(* IEC 61131-3 sources: AXOpen/src/components.dukane.welders/ctrl/src/Axo_IQ_SeriesWelder (part 6) *)

                    IF TRUE THEN
                        THIS.CallTimers(FALSE);
                        _progress := 474;
                    END_IF;
                END_IF;

                IF _progress = 474 THEN                                                                                     // TemplateTask_20steps_6 running: , <add the detailed description of the current action 15>
                    IF _infoTimer.output THEN
                        TaskMessenger.Activate( UINT#674, eAxoMessageCategory#Warning);
                        Status.Error.Id :=      UINT#674;
                    END_IF;

                    IF TRUE THEN
                        THIS.CallTimers(FALSE);
                        _progress := 475;
                    END_IF;
                END_IF;

                IF _progress = 475 THEN                                                                                     // TemplateTask_20steps_6 running: , <add the detailed description of the current action 16>
                    IF _infoTimer.output THEN
                        TaskMessenger.Activate( UINT#675, eAxoMessageCategory#Warning);
                        Status.Error.Id :=      UINT#675;
                    END_IF;

                    IF TRUE THEN
                        THIS.CallTimers(FALSE);
                        _progress := 476;
                    END_IF;
                END_IF;

                IF _progress = 476 THEN                                                                                     // TemplateTask_20steps_6 running: , <add the detailed description of the current action 17>
                    IF _infoTimer.output THEN
                        TaskMessenger.Activate( UINT#676, eAxoMessageCategory#Warning);
                        Status.Error.Id :=      UINT#676;
                    END_IF;

                    IF TRUE THEN
                        THIS.CallTimers(FALSE);
                        _progress := 477;
                    END_IF;
                END_IF;

                IF _progress = 477 THEN                                                                                     // TemplateTask_20steps_6 running: , <add the detailed description of the current action 18>
                    IF _infoTimer.output THEN
                        TaskMessenger.Activate( UINT#677, eAxoMessageCategory#Warning);
                        Status.Error.Id :=      UINT#677;
                    END_IF;

                    IF TRUE THEN
                        THIS.CallTimers(FALSE);
                        _progress := 478;
                    END_IF;
                END_IF;

                IF _progress = 478 THEN                                                                                     // TemplateTask_20steps_6 running: , <add the detailed description of the current action 19>
                    IF _infoTimer.output THEN
                        TaskMessenger.Activate( UINT#678, eAxoMessageCategory#Warning);
                        Status.Error.Id :=      UINT#678;
                    END_IF;

                    IF TRUE THEN
                        THIS.CallTimers(FALSE);
                        _progress := 479;
                    END_IF;
                END_IF;

                IF _progress = 479 THEN                                                                                     // TemplateTask_20steps_6 running: , <add the detailed description of the current action 20>
                    TemplateTask_20steps_6.DoneWhen(TRUE);
                    _progress := 0;
                END_IF;

                THIS.CallTimers(TRUE);

                TemplateTask_20steps_6.ThrowWhen(_errorTimer.output);
                Status.Action.Id := TO_UINT(_progress);
                TemplateTask_20steps_6.ThrowWhen(TemplateTask_20steps_6.Duration >= Config.TaskTimeout AND Config.TaskTimeout > T#0s ,'TemplateTask_20steps_6 timeout.');
            END_IF;
            IF TemplateTask_20steps_6.DoneReached() THEN
                Status.Action.Id :=  UINT#261;
                Status.Error.Id :=  UINT#0;
            ELSIF TemplateTask_20steps_6.ErrorOccured() THEN
                Status.Action.Id :=  UINT#10160;
                Status.Error.Id  :=  UINT#10160;
            ELSIF TemplateTask_20steps_6.AbortTriggered()THEN
                Status.Action.Id :=  UINT#10161;
                Status.Error.Id  :=  UINT#10161;
            END_IF;
            Messenger.ActivateOnCondition(ULINT#10160,TemplateTask_20steps_6.HasError(), eAxoMessageCategory#Error);
            Messenger.ActivateOnCondition(ULINT#10161,TemplateTask_20steps_6.IsAborted(), eAxoMessageCategory#Error);
            Messenger.ActivateOnCondition(ULINT#262,TemplateTask_20steps_6.RestoreTriggered() , eAxoMessageCategory#Error);
            IF TemplateTask_20steps_6.RestoreTriggered() AND _progress >= 460 AND _progress <= 479  THEN
                Status.Action.Id :=  UINT#262;
                _progress := 0;
            END_IF;
            //******************************************

            //***********Update outputs ****************
            // ============================================================================
            // Network 14: Write synchronous data to the module (outputs)
            // ============================================================================
            // This was original outputs writing =>
            // synchronous_write_retval := DPWR_DAT(LADDR := outputs_hw_id,RECORD := iq_if._out);
            // <= This was original outputs writing

            // This is new outputs writing =>
            _data_out[0].%X0    :=  Outputs.N0;
            _data_out[0].%X1    :=  Outputs.N01;
            _data_out[0].%X2    :=  Outputs.N02;
            _data_out[0].%X3    :=  Outputs.N03;
            _data_out[0].%X4    :=  Outputs.N04;
            _data_out[0].%X5    :=  Outputs.N05;
            _data_out[0].%X6    :=  Outputs.N06;
            _data_out[0].%X7    :=  Outputs.ClearSetup;
            _data_out[1].%X0    :=  Outputs.N2;
            _data_out[1].%X1    :=  Outputs.N3;
            _data_out[1].%X2    :=  Outputs.N4;
            _data_out[1].%X3    :=  Outputs.N5;
            _data_out[1].%X4    :=  Outputs.N6;
            _data_out[1].%X5    :=  Outputs.N7;
            _data_out[1].%X6    :=  Outputs.N8;
            _data_out[1].%X7    :=  Outputs.N9;
            _data_out[2].%X0    :=  Outputs.RunScan;
            _data_out[2].%X1    :=  Outputs.N11;
            _data_out[2].%X2    :=  Outputs.N12;
            _data_out[2].%X3    :=  Outputs.N13;
            _data_out[2].%X4    :=  Outputs.N14;
            _data_out[2].%X5    :=  Outputs.N15;
            _data_out[2].%X6    :=  Outputs.N16;
            _data_out[2].%X7    :=  Outputs.N17;
            _data_out[3].%X0    :=  Outputs.RunContinuously;
            _data_out[3].%X1    :=  Outputs.RunWeld;
            _data_out[3].%X2    :=  Outputs.RunTest;
            _data_out[3].%X3    :=  Outputs.ClearError;
            _data_out[3].%X4    :=  Outputs.OTF_AmplitudeEnable;
            _data_out[3].%X5    :=  Outputs.CycleStop;
            _data_out[3].%X6    :=  Outputs.FrontPanelLockout_0;
            _data_out[3].%X7    :=  Outputs.FrontPanelLockout_1;

            tmp_DW              :=  TO_DWORD(Outputs.OTF_Amp_Setpoint);
            _data_out[4]        :=  tmp_DW.%B3;
            _data_out[5]        :=  tmp_DW.%B2;
            _data_out[6]        :=  tmp_DW.%B1;
            _data_out[7]        :=  tmp_DW.%B0;

            tmp_DW              :=  TO_DWORD(Outputs.ActiveSetupSelection);
            _data_out[8]        :=  tmp_DW.%B3;
            _data_out[9]        :=  tmp_DW.%B2;
            _data_out[10]       :=  tmp_DW.%B1;
            _data_out[11]       :=  tmp_DW.%B0;

            tmp_DW              :=  TO_DWORD(Outputs.RunningSetupSelection);
            _data_out[12]       :=  tmp_DW.%B3;
            _data_out[13]       :=  tmp_DW.%B2;
            _data_out[14]       :=  tmp_DW.%B1;
            _data_out[15]       :=  tmp_DW.%B0;

            tmp_DW              :=  TO_DWORD(Outputs.RunningMPCProbeSelection);
            _data_out[16]       :=  tmp_DW.%B3;
            _data_out[17]       :=  tmp_DW.%B2;
            _data_out[18]       :=  tmp_DW.%B1;
            _data_out[19]       :=  tmp_DW.%B0;

            synchronous_write_retval := TO_INT(WriteData(LADDR := TO_WORD(Config.HWIDs.HwID_PLC_to_iQ_Outputs),RECORD := _data_out));
            IF synchronous_write_retval > INT#0 THEN
                Messenger.Activate(UINT#1231, eAxoMessageCategory#ProgrammingError);
                Status.Error.Id := UINT#1231;
                RETURN;
            END_IF;
            // <= This is new outputs writing

            // ============================================================================
            // Network 15: Read req - HMI export (indicators)
            // ============================================================================
            // tof_async_read_ind(IN := (par_read_map <> 0) OR (on_demand_read_map <> 0) OR (model_read_map <> 0),PT := T#500ms);
            // Hmi.s.AsyncReadIndicator := tof_async_read_ind.Q;
            tof_async_read_ind(signal := (par_read_map <> WORD#0) OR (on_demand_read_map <> WORD#0) OR (model_read_map <> WORD#0) , duration := T#500ms);
            Hmi.s.AsyncReadIndicator := tof_async_read_ind.output;

            // ============================================================================
            // Network 16: Read acyclic data
            // ============================================================================
            //Try asynchronous comunication only when synchronous comunication is stable (no errors for 1s)
            // IF (coms_stable) THEN

            //     //Save rd_req value from previous iteation
            //     prev_rd_req := ReadRecord.request;

            //     // Proces valid data if needed
            //     IF ReadRecord.VALID THEN
            //         Hmi.read_status[async_read_no] := ReadRecord.STATUS;
            //         CASE async_read_no OF
            //             -16: // Model no decode to string
            //                 // Chars_TO_Strg(Chars := str_read_buffer,
            //                 //               pChars := 0,
            //                 //               Cnt := RD_REC.length,
            //                 //               Strg => ModelInfo.ModelNumber);
            //                 _data_255[0]:= TO_BYTE(ReadRecord.length);
            //                 FOR index := UINT#0 TO ReadRecord.length DO
            //                     _data_255[index + UINT#1] := str_read_buffer_254[index];
            //                 END_FOR;
            //                 Deserialize(UDINT#0, str_read_buffer_254, ModelInfo.ModelNumber);

            //             -15:
            //                 Deserialize(UDINT#0, str_read_buffer_254, ModelInfo.SerialNumber);

            //             -14: // MB firmware version decode to string
            //                 // Chars_TO_Strg(Chars := str_read_buffer_254,
            //                 //               pChars := 0,
            //                 //               Cnt := RD_REC.length,
            //                 //               Strg => ModelInfo.MB_FirmwareVersion);
            //                 _data_255[0]:= TO_BYTE(ReadRecord.length);
            //                 FOR index := UINT#0 TO ReadRecord.length DO
            //                     _data_255[index + UINT#1] := str_read_buffer_254[index];
            //                 END_FOR;
            //                 Deserialize(UDINT#0, str_read_buffer_254, ModelInfo.MB_FirmwareVersion);

            //             -13: // FP firmware version decode to string
            //                 // Chars_TO_Strg(Chars := str_read_buffer_254,
            //                 //               pChars := 0,
            //                 //               Cnt := RD_REC.length,
            //                 //               Strg => ModelInfo.FP_FirmwareVersion);
            //                 _data_255[0]:= TO_BYTE(ReadRecord.length);
            //                 FOR index := UINT#0 TO ReadRecord.length DO
            //                     _data_255[index + UINT#1] := str_read_buffer_254[index];
            //                 END_FOR;
            //                 Deserialize(UDINT#0, str_read_buffer_254, ModelInfo.FP_FirmwareVersion);

            //             -12: // MB bootloader version decode to string
            //                 // Chars_TO_Strg(Chars := str_read_buffer_254,
            //                 //               pChars := 0,
            //                 //               Cnt := RD_REC.length,
            //                 //               Strg => ModelInfo.MB_BootLoaderVersion);
            //                 _data_255[0]:= TO_BYTE(ReadRecord.length);
            //                 FOR index := UINT#0 TO ReadRecord.length DO
            //                     _data_255[index + UINT#1] := str_read_buffer_254[index];
            //                 END_FOR;
            //                 Deserialize(UDINT#0, str_read_buffer_254, ModelInfo.MB_BootLoaderVersion);

            //             -11: // FP bootloader version decode to string
            //                 // Chars_TO_Strg(Chars := str_read_buffer_254,
            //                 //               pChars := 0,
            //                 //               Cnt := RD_REC.length,
            //                 //               Strg => ModelInfo.FP_BootloaderVersion);
            //                 _data_255[0]:= TO_BYTE(ReadRecord.length);
            //                 FOR index := UINT#0 TO ReadRecord.length DO
            //                     _data_255[index + UINT#1] := str_read_buffer_254[index];
            //                 END_FOR;
            //                 Deserialize(UDINT#0, str_read_buffer_254, ModelInfo.FP_BootloaderVersion);

            //             1:  //Data 1 read to buffer succesfull - copy
            //                 Parameters.ProcCtrl := ReadBuffers.buf1.ProcCtrl;
            //                 Parameters.ProcLimits := ReadBuffers.buf1.ProcLimits;
            //                 Parameters.FreqCtrl := ReadBuffers.buf1.FreqCtrl;
            //                 Parameters.TriggerByPower := ReadBuffers.buf1.TriggerByPower;
            //                 Parameters.FreqCtrlMode := ReadBuffers.buf1.FreqCtrlMode;

            //             2: //Data 2 read to buffer succesfull - copy
            //                 Parameters.PowerReg := ReadBuffers.buf2.PowerReg;
            //                 Parameters.PressPretrigger := ReadBuffers.buf2.PressPretrigger;
            //                 Parameters.PressTrigger := ReadBuffers.buf2.PressTrigger;
            //                 Parameters.PressTriggerDelay := ReadBuffers.buf2.PressTriggerDelay;
            //                 Parameters.PressWeld := ReadBuffers.buf2.PressWeld;
            //                 Parameters.PressWeldScrub := ReadBuffers.buf2.PressWeldScrub;
            //                 Parameters.PressPostWeld := ReadBuffers.buf2.PressPostWeld;
            //             3: //Data 3 read to buffer succesfull - copy
            //                 Parameters.PressLimits.TriggerTime := ReadBuffers.buf3.TriggerTime;
            //                 Parameters.PressLimits.TriggerPosition := ReadBuffers.buf3.TriggerPosition;
            //                 Parameters.PressLimits.TriggerDelayTime := ReadBuffers.buf3.TriggerDelayTime;
            //                 Parameters.PressLimits.TriggerDelayDistance := ReadBuffers.buf3.TriggerDelayDistance;
            //                 Parameters.PressLimits.Weld1Distance := ReadBuffers.buf3.Weld1Distance;
            //                 Parameters.PressLimits.Weld1Position := ReadBuffers.buf3.Weld1Position;
            //                 Parameters.PressLimits.Weld2Time := ReadBuffers.buf3.Weld2Time;
            //                 Parameters.PressLimits.Weld2Energy := ReadBuffers.buf3.Weld2Energy;
            //                 Parameters.PressLimits.Weld2Power := ReadBuffers.buf3.Weld2Power;
            //             4: //Data 4 read to buffer succesfull - copy
            //                 Parameters.PressLimits.Weld2Distance := ReadBuffers.buf4.Weld2Distance;
            //                 Parameters.PressLimits.Weld2Position := ReadBuffers.buf4.Weld2Position;
            //                 Parameters.PressLimits.TotalWeldTime := ReadBuffers.buf4.TotalWeldTime;
            //                 Parameters.PressLimits.TotalWeldEnergy := ReadBuffers.buf4.TotalWeldEnergy;
            //                 Parameters.PressLimits.TotalWeldDistance := ReadBuffers.buf4.TotalWeldDistance;
            //                 Parameters.PressLimits.DynamicHoldTime := ReadBuffers.buf4.DynamicHoldTime;
            //                 Parameters.PressLimits.DynamicHoldDistance := ReadBuffers.buf4.DynamicHoldDistance;
            //                 Parameters.PressLimits.TotalCycleTime := ReadBuffers.buf4.TotalCycleTime;
            //                 Parameters.PressLimits.FinalHoldPosition := ReadBuffers.buf4.FinalHoldPosition;
            //                 Parameters.PressLimits.ErrorStatus := ReadBuffers.buf4.ErrorStatus;
            //             5: //Data 5 read to buffer succesfull - copy
            //                 Parameters.AnalogSensor := ReadBuffers.buf5.AnalogSensor;
            //                 Parameters.AfterburstEnable := ReadBuffers.buf5.AfterburstEnable;
            //                 Parameters.LimitWeld1TimeEnable := ReadBuffers.buf5.LimitWeld1TimeEnable;
            //                 Parameters.LimitWeld1EnergyEnable := ReadBuffers.buf5.LimitWeld1EnergyEnable;
            //                 Parameters.LimitWeld1PowerEnable := ReadBuffers.buf5.LimitWeld1PowerEnable;
            //             17://Test scan read finished succesfully
            //                 Hmi.s.DisplayApplyScannedFrequency := true;

            //         END_CASE;
            //     END_IF;

            //     // Read request error - reset invalidated date if needed
            //     IF ReadRecord.ERROR THEN
            //         Hmi.read_status[async_read_no] := ReadRecord.STATUS;

            //         CASE async_read_no OF
            //             -16:
            //                 ModelInfo.ModelNumber := '';
            //             -15:
            //                 ModelInfo.SerialNumber := 0;
            //             -14:
            //                 ModelInfo.MB_FirmwareVersion := '';
            //             -13:
            //                 ModelInfo.FP_FirmwareVersion := '';
            //             -12:
            //                 ModelInfo.MB_BootLoaderVersion := '';
            //             -11:
            //                 ModelInfo.FP_BootloaderVersion := '';
            //         END_CASE;
            //     END_IF;

            //     // Unmask bit map after successfully / unsuccesfully finished readout of model no
            //     IF (ReadRecord.VALID OR ReadRecord.ERROR) THEN
            //         IF (async_read_no < 0) AND (async_read_no >= -16) THEN
            //             mask := THIS.DECO_WORD(TO_UINT(async_read_no + 16));
            //             model_read_map := model_read_map AND (NOT mask);
            //         END_IF;

            //         IF (async_read_no > 13) AND (async_read_no < + 32) THEN
            //             mask := THIS.DECO_WORD(TO_UINT(async_read_no - 17));
            //             on_demand_read_map := on_demand_read_map AND (NOT mask);
            //         END_IF;
            //     END_IF;

            //     // Unmask bit map after successfully finished readout of parameters
            //     IF ReadRecord.VALID THEN
            //         IF (async_read_no > 0) AND (async_read_no <= 16) THEN
            //             mask := THIS.DECO_WORD(TO_UINT(async_read_no - 1));
            //             par_read_map := par_read_map AND (NOT mask);
            //         END_IF;
            //     END_IF;

            //     rd_any_response := (ReadRecord.BUSY OR ReadRecord.VALID OR ReadRecord.ERROR);

            //     //If we get a signal that request was processed we can set it to false to prepare for generating a new rising edge
            //     IF rd_req AND rd_any_response THEN
            //         rd_req := false;
            //     END_IF;

            //     //If the previous request was processed and we are ready for a new one (new rising edge on rd_req) lets create one
            //     IF (NOT prev_rd_req) AND (NOT rd_any_response) AND (NOT coms_just_restored) THEN
            //         IF (model_read_map <> WORD#0) THEN
            //             async_read_no := THIS.ENCO(model_read_map) - INT#16;
            //             rd_req := true;
            //         ELSIF (on_demand_read_map <> WORD#0) THEN
            //             async_read_no := THIS.ENCO(on_demand_read_map) + INT#17;
            //             rd_req := true;
            //         ELSIF (par_read_map <> WORD#0) THEN
            //             async_read_no := THIS.ENCO(par_read_map) + INT#1;
            //             rd_req := true;
            //         ELSE
            //             //If no request present we call the default RD_REC but without request
            //             async_read_no := 0;
            //         END_IF;
            //     END_IF;

            //     //Perform the read itself
            //     CASE async_read_no OF
            //         -16: //Read model no string
            //             ReadRecord( request := rd_req,
            //                     id := TO_WORD(Config.HWIDs.HwID_iQ_to_PLC_Inputs),
            //                     index := index_async_model_no,
            //                     maxLength := UINT#64,
            //                     record := str_read_buffer_254);
            //         -15:  //Read serial no
            //             ReadRecord( request := rd_req,
            //                     id := TO_WORD(Config.HWIDs.HwID_iQ_to_PLC_Inputs),
            //                     index := index_async_serial_no,
            //                     maxLength := UINT#4,
            //                     record :=  str_read_buffer_254); // ModelInfo.SerialNumber);
            //         -14: //Read mb firmware version
            //             ReadRecord( request := rd_req,
            //                     id := TO_WORD(Config.HWIDs.HwID_iQ_to_PLC_Inputs),
            //                     index := index_async_mb_firmware_ver,
            //                     maxLength := UINT#64,
            //                     record := str_read_buffer_254);
            //         -13: //Read fp firmware version
            //             ReadRecord( request := rd_req,
            //                     id := TO_WORD(Config.HWIDs.HwID_iQ_to_PLC_Inputs),
            //                     index := index_async_fp_firmware_ver,
            //                     maxLength := UINT#64,
            //                     record := str_read_buffer_254);
            //         -12: //Read mb bootloader version
            //             ReadRecord( request := rd_req,
            //                     id := TO_WORD(Config.HWIDs.HwID_iQ_to_PLC_Inputs),
            //                     index := index_async_mb_bootloader_no,
            //                     maxLength := UINT#64,
            //                     record := str_read_buffer_254);
            //         -11: //Read fp bootloader version
            //             ReadRecord( request := rd_req,
            //                     id := TO_WORD(Config.HWIDs.HwID_iQ_to_PLC_Inputs),
            //                     index := index_async_fp_bootloader_no,
            //                     maxLength := UINT#64,
            //                     record := str_read_buffer_254);

            //         1:  //Read parameter packet 1
            //             ReadRecord( request := rd_req,
            //                     id := TO_WORD(Config.HWIDs.HwID_iQ_to_PLC_Inputs),
            //                     index := index_async_data1,
            //                     maxLength := UINT#132,
            //                     record := str_read_buffer_254);
            //                     THIS.ByteArray_TO_buf1(str_read_buffer_254,ReadBuffers.buf1);
            //         2:  //Read parameter packet 2
            //             ReadRecord( request := rd_req,
            //                     id := TO_WORD(Config.HWIDs.HwID_iQ_to_PLC_Inputs),
            //                     index := index_async_data2,
            //                     maxLength := UINT#136,
            //                     record := str_read_buffer_254);
            //                     THIS.ByteArray_TO_buf2(str_read_buffer_254,ReadBuffers.buf2);
            //         3:  //Read parameter packet 3
            //             ReadRecord( request := rd_req,
            //                     id := TO_WORD(Config.HWIDs.HwID_iQ_to_PLC_Inputs),
            //                     index := index_async_data3,
            //                     maxLength := UINT#180,
            //                     record := str_read_buffer_254);
            //                     THIS.ByteArray_TO_buf3(str_read_buffer_254,ReadBuffers.buf3);
            //         4:  //Read parameter packet 4
            //             ReadRecord( request := rd_req,
            //                     id := TO_WORD(Config.HWIDs.HwID_iQ_to_PLC_Inputs),
            //                     index := index_async_data4,
            //                     maxLength := UINT#200,
            //                     record := str_read_buffer_254);
            //                     THIS.ByteArray_TO_buf4(str_read_buffer_254,ReadBuffers.buf4);
            //         5:  //Read parameter packet 5
            //             ReadRecord( request := rd_req,
            //                     id := TO_WORD(Config.HWIDs.HwID_iQ_to_PLC_Inputs),
            //                     index := index_async_data5,
            //                     maxLength := UINT#176,
            //                     record := str_read_buffer_254);
            //                     THIS.ByteArray_TO_buf5(str_read_buffer_254,ReadBuffers.buf5);

            //             //Start of on-demand request types
            //         17: //Read test scan results
            //             ReadRecord( request := rd_req,
            //                     id := TO_WORD(Config.HWIDs.HwID_iQ_to_PLC_Inputs),
            //                     index := index_async_test_scan_result,
            //                     maxLength := UINT#4,
            //                     record := str_read_buffer_254);
            //                     TestScanResults.TestScanResults:=       TO_DINT(SHL(TO_DWORD(str_read_buffer_254[  0]), UINT#24) OR
            //                                                                             SHL(TO_DWORD(str_read_buffer_254[  1]), UINT#16) OR
            //                                                                             SHL(TO_DWORD(str_read_buffer_254[  2]),  UINT#8) OR
            //                                                                                 TO_DWORD(str_read_buffer_254[  3]));
            //         ELSE
            //             //By default we call test scan results request (but req is off so o data transfer)
            //             ReadRecord( request := FALSE,
            //                     id := TO_WORD(Config.HWIDs.HwID_iQ_to_PLC_Inputs),
            //                     index := index_async_test_scan_result,
            //                     maxLength := UINT#4,
            //                     record := str_read_buffer_254);
            //                     TestScanResults.TestScanResults:=       TO_DINT(SHL(TO_DWORD(str_read_buffer_254[  0]), UINT#24) OR
            //                                                                             SHL(TO_DWORD(str_read_buffer_254[  1]), UINT#16) OR
            //                                                                             SHL(TO_DWORD(str_read_buffer_254[  2]),  UINT#8) OR
            //                                                                                 TO_DWORD(str_read_buffer_254[  3]));
            //     END_CASE;

            // END_IF;

            // ============================================================================
            // Network 17: Analog sensor settings HMI processing
            // ============================================================================
            // // Currently supports only distance / MPC distance modes
            // IF Hmi.c.selected_analog_sensor > 8 THEN
            //     Hmi.c.selected_analog_sensor := 8;
            // ELSIF Hmi.c.selected_analog_sensor < 1 THEN
            //     Hmi.c.selected_analog_sensor := 1;
            // END_IF;

            // tmp_W := par_read_map AND TO_WORD(2#0000000000010000);
            // IF tmp_W <> WORD#0 THEN
            //     Hmi.s.current_analog_sensor := 0;
            // END_IF;

            // IF coms_stable THEN
            //     IF Hmi.analog_sensor_data.Enable >= 2 THEN
            //         IF Inputs.SystemStatus.MPC_Present THEN
            //             Hmi.analog_sensor_data.Enable := 3;
            //         ELSE
            //             Hmi.analog_sensor_data.Enable := 2;
            //         END_IF;
            //     ELSE
            //         Hmi.analog_sensor_data.Enable := 0;
            //     END_IF;
            // END_IF;

            // IF coms_stable AND par_read_map = WORD#0 THEN
            //     IF Hmi.c.selected_analog_sensor <> Hmi.s.current_analog_sensor THEN
            //         Hmi.analog_sensor_data := Parameters.AnalogSensor.Sensor[Hmi.c.selected_analog_sensor];
            //         Hmi.s.current_analog_sensor := Hmi.c.selected_analog_sensor;
            //         IF Inputs.SystemStatus.MPC_Present THEN
            //             Hmi.c.selected_analog_sensor := Hmi.c.selected_analog_sensor;
            //         END_IF;
            //     ELSE
            //     //  IF Parameters.AnalogSensor.Sensor[Hmi.c.selected_analog_sensor] <> Hmi.analog_sensor_data THEN
            //         IF THIS.AnalogSensorDiffers(REF(Parameters.AnalogSensor.Sensor[Hmi.c.selected_analog_sensor]) , REF(Hmi.analog_sensor_data)) THEN
            //             Parameters.AnalogSensor.Sensor[Hmi.c.selected_analog_sensor] := Hmi.analog_sensor_data;
            //         END_IF;
            //     END_IF;
            //     IF NOT Inputs.SystemStatus.MPC_Present THEN
            //         Outputs.RunningMPCProbeSelection := 0;
            //     END_IF;
            // END_IF;

            // ============================================================================
            // Network 18: Trigger writes on user data change
            // ============================================================================

            // //Posibly compare only in certain cycles to limit the large data block comparison PLC load (if multiple IQ installed)
            // IF AxoTaskCompareThisCycle THEN
            //     // We can only triger writes if we have communication and all parameters were already read
            //     IF (Config_async_write_permited AND coms_stable AND (NOT coms_just_restored) AND (par_read_map = WORD#0)) THEN
            //         IF (comp_opt_cycler = 0) THEN
            //             // IF (Parameters.ProcCtrl <> ReadBuffers.buf1.ProcCtrl) OR
            //             //     (Parameters.ProcLimits <> ReadBuffers.buf1.ProcLimits) OR
            //             //     (Parameters.FreqCtrl <> ReadBuffers.buf1.FreqCtrl) OR
            //             //     (Parameters.TriggerByPower <> ReadBuffers.buf1.TriggerByPower) OR
            //             //     (Parameters.FreqCtrlMode <> ReadBuffers.buf1.FreqCtrlMode) THEN
            //             IF  (THIS.ProcCtrlDiffers(       REF(Parameters.ProcCtrl)       , REF(ReadBuffers.buf1.ProcCtrl)))       OR
            //                 (THIS.ProcLimitsDiffers(     REF(Parameters.ProcLimits)     , REF(ReadBuffers.buf1.ProcLimits)))     OR
            //                 (THIS.FreqCtrlDiffers(       REF(Parameters.FreqCtrl)       , REF(ReadBuffers.buf1.FreqCtrl)))       OR
            //                 (THIS.TriggerByPowerDiffers( REF(Parameters.TriggerByPower) , REF(ReadBuffers.buf1.TriggerByPower))) OR
            //                 (Parameters.FreqCtrlMode <> ReadBuffers.buf1.FreqCtrlMode) THEN
            //                     par_write_map := par_write_map OR TO_WORD(2#000000000000001);
            //             END_IF;
            //         END_IF;
            //         IF (comp_opt_cycler = 1) THEN
            //             // IF (Parameters.PowerReg <> ReadBuffers.buf2.PowerReg) OR
            //             //     (Parameters.PressPretrigger <> ReadBuffers.buf2.PressPretrigger) OR
            //             //     (Parameters.PressTrigger <> ReadBuffers.buf2.PressTrigger) OR
            //             //     (Parameters.PressTriggerDelay <> ReadBuffers.buf2.PressTriggerDelay) OR
            //             //     (Parameters.PressWeld <> ReadBuffers.buf2.PressWeld) OR
            //             //     (Parameters.PressWeldScrub <> ReadBuffers.buf2.PressWeldScrub) OR
            //             //     (Parameters.PressPostWeld <> ReadBuffers.buf2.PressPostWeld) THEN
            //             IF  (THIS.PowerRegDiffers(          REF(Parameters.PowerReg)           ,   REF(ReadBuffers.buf2.PowerReg))) OR
            //                 (THIS.PressPretriggerDiffers(   REF(Parameters.PressPretrigger)    ,   REF(ReadBuffers.buf2.PressPretrigger))) OR
            //                 (THIS.PressTriggerDiffers(      REF(Parameters.PressTrigger)       ,   REF(ReadBuffers.buf2.PressTrigger))) OR
            //                 (THIS.PressTriggerDelayDiffers( REF(Parameters.PressTriggerDelay)  ,   REF(ReadBuffers.buf2.PressTriggerDelay))) OR
            //                 (THIS.PressWeldDiffers(         REF(Parameters.PressWeld)          ,   REF(ReadBuffers.buf2.PressWeld))) OR
            //                 (THIS.PressWeldScrubDiffers(    REF(Parameters.PressWeldScrub)     ,   REF(ReadBuffers.buf2.PressWeldScrub))) OR
            //                 (THIS.PressPostWeldDiffers(     REF(Parameters.PressPostWeld)      ,   REF(ReadBuffers.buf2.PressPostWeld))) THEN
            //                 par_write_map := par_write_map OR TO_WORD(2#000000000000010);
            //             END_IF;
            //         END_IF;
            //         IF (comp_opt_cycler = 2) THEN
            //             // IF (Parameters.PressLimits.TriggerTime <> ReadBuffers.buf3.TriggerTime) OR
            //             //     (Parameters.PressLimits.TriggerPosition <> ReadBuffers.buf3.TriggerPosition) OR
            //             //     (Parameters.PressLimits.TriggerDelayTime <> ReadBuffers.buf3.TriggerDelayTime) OR
            //             //     (Parameters.PressLimits.TriggerDelayDistance <> ReadBuffers.buf3.TriggerDelayDistance) OR
            //             //     (Parameters.PressLimits.Weld1Distance <> ReadBuffers.buf3.Weld1Distance) OR
            //             //     (Parameters.PressLimits.Weld1Position <> ReadBuffers.buf3.Weld1Position) OR
            //             //     (Parameters.PressLimits.Weld2Time <> ReadBuffers.buf3.Weld2Time) OR
            //             //     (Parameters.PressLimits.Weld2Energy <> ReadBuffers.buf3.Weld2Energy) OR
            //             //     (Parameters.PressLimits.Weld2Power <> ReadBuffers.buf3.Weld2Power) THEN
            //             IF  (THIS.PressLimitDiffers(REF(Parameters.PressLimits.TriggerTime)            ,   REF( ReadBuffers.buf3.TriggerTime))) OR
            //                 (THIS.PressLimitDiffers(REF(Parameters.PressLimits.TriggerPosition)        ,   REF( ReadBuffers.buf3.TriggerPosition))) OR
            //                 (THIS.PressLimitDiffers(REF(Parameters.PressLimits.TriggerDelayTime)       ,   REF( ReadBuffers.buf3.TriggerDelayTime))) OR
            //                 (THIS.PressLimitDiffers(REF(Parameters.PressLimits.TriggerDelayDistance)   ,   REF( ReadBuffers.buf3.TriggerDelayDistance))) OR
            //                 (THIS.PressLimitDiffers(REF(Parameters.PressLimits.Weld1Distance)          ,   REF( ReadBuffers.buf3.Weld1Distance))) OR
            //                 (THIS.PressLimitDiffers(REF(Parameters.PressLimits.Weld1Position)          ,   REF( ReadBuffers.buf3.Weld1Position))) OR
            //                 (THIS.PressLimitDiffers(REF(Parameters.PressLimits.Weld2Time)              ,   REF( ReadBuffers.buf3.Weld2Time))) OR
            //                 (THIS.PressLimitDiffers(REF(Parameters.PressLimits.Weld2Energy)            ,   REF( ReadBuffers.buf3.Weld2Energy))) OR
            //                 (THIS.PressLimitDiffers(REF(Parameters.PressLimits.Weld2Power)             ,   REF( ReadBuffers.buf3.Weld2Power))) THEN
            //                 par_write_map := par_write_map OR TO_WORD(2#000000000000100);
            //             END_IF;
            //         END_IF;
            //         IF (comp_opt_cycler = 3) THEN
            //             // IF (Parameters.PressLimits.Weld2Distance <> ReadBuffers.buf4.Weld2Distance) OR
            //             //     (Parameters.PressLimits.Weld2Position <> ReadBuffers.buf4.Weld2Position) OR
            //             //     (Parameters.PressLimits.TotalWeldTime <> ReadBuffers.buf4.TotalWeldTime) OR
            //             //     (Parameters.PressLimits.TotalWeldEnergy <> ReadBuffers.buf4.TotalWeldEnergy) OR
            //             //     (Parameters.PressLimits.TotalWeldDistance <> ReadBuffers.buf4.TotalWeldDistance) OR
            //             //     (Parameters.PressLimits.DynamicHoldTime <> ReadBuffers.buf4.DynamicHoldTime) OR
            //             //     (Parameters.PressLimits.DynamicHoldDistance <> ReadBuffers.buf4.DynamicHoldDistance) OR
            //             //     (Parameters.PressLimits.TotalCycleTime <> ReadBuffers.buf4.TotalCycleTime) OR
            //             //     (Parameters.PressLimits.FinalHoldPosition <> ReadBuffers.buf4.FinalHoldPosition) OR
            //             //     (Parameters.PressLimits.ErrorStatus <> ReadBuffers.buf4.ErrorStatus) THEN
            //             IF  (THIS.PressLimitDiffers(REF(Parameters.PressLimits.Weld2Distance)          ,   REF(ReadBuffers.buf4.Weld2Distance))) OR
            //                 (THIS.PressLimitDiffers(REF(Parameters.PressLimits.Weld2Position)          ,   REF(ReadBuffers.buf4.Weld2Position))) OR
            //                 (THIS.PressLimitDiffers(REF(Parameters.PressLimits.TotalWeldTime)          ,   REF(ReadBuffers.buf4.TotalWeldTime))) OR
            //                 (THIS.PressLimitDiffers(REF(Parameters.PressLimits.TotalWeldEnergy)        ,   REF(ReadBuffers.buf4.TotalWeldEnergy))) OR
            //                 (THIS.PressLimitDiffers(REF(Parameters.PressLimits.TotalWeldDistance)      ,   REF(ReadBuffers.buf4.TotalWeldDistance))) OR
            //                 (THIS.PressLimitDiffers(REF(Parameters.PressLimits.DynamicHoldTime)        ,   REF(ReadBuffers.buf4.DynamicHoldTime))) OR
            //                 (THIS.PressLimitDiffers(REF(Parameters.PressLimits.DynamicHoldDistance)    ,   REF(ReadBuffers.buf4.DynamicHoldDistance))) OR
            //                 (THIS.PressLimitDiffers(REF(Parameters.PressLimits.TotalCycleTime)         ,   REF(ReadBuffers.buf4.TotalCycleTime))) OR
            //                 (THIS.PressLimitDiffers(REF(Parameters.PressLimits.FinalHoldPosition)      ,   REF(ReadBuffers.buf4.FinalHoldPosition))) OR
            //                 (THIS.PressLimitDiffers(REF(Parameters.PressLimits.ErrorStatus)            ,   REF(ReadBuffers.buf4.ErrorStatus))) THEN
            //                     par_write_map := par_write_map OR TO_WORD(2#000000000001000);
            //             END_IF;
            //         END_IF;
            //         IF (comp_opt_cycler = 4) THEN
            //             // IF (Parameters.AnalogSensor <> ReadBuffers.buf5.AnalogSensor) OR
            //             //     (Parameters.AfterburstEnable <> ReadBuffers.buf5.AfterburstEnable) OR
            //             //     (Parameters.LimitWeld1TimeEnable <> ReadBuffers.buf5.LimitWeld1TimeEnable) OR
            //             //     (Parameters.LimitWeld1EnergyEnable <> ReadBuffers.buf5.LimitWeld1EnergyEnable) OR
            //             //     (Parameters.LimitWeld1PowerEnable <> ReadBuffers.buf5.LimitWeld1PowerEnable) THEN
            //             IF  (THIS.AnalogSensorSpecDiffers(REF(Parameters.AnalogSensor)             ,   REF(ReadBuffers.buf5.AnalogSensor))) OR
            //                 (Parameters.AfterburstEnable                                           <>  ReadBuffers.buf5.AfterburstEnable) OR
            //                 (THIS.PressLimitEnableDiffers(REF(Parameters.LimitWeld1TimeEnable)     ,   REF( ReadBuffers.buf5.LimitWeld1TimeEnable))) OR
            //                 (THIS.PressLimitEnableDiffers(REF(Parameters.LimitWeld1EnergyEnable)   ,   REF( ReadBuffers.buf5.LimitWeld1EnergyEnable))) OR
            //                 (THIS.PressLimitEnableDiffers(REF(Parameters.LimitWeld1PowerEnable)    ,   REF( ReadBuffers.buf5.LimitWeld1PowerEnable))) THEN
            //                 par_write_map := par_write_map OR TO_WORD(2#000000000010000);
            //             END_IF;
            //         END_IF;
            //         comp_opt_cycler := (comp_opt_cycler + 1) MOD 5;
            //     END_IF;
            // END_IF;

            // ============================================================================
            // Network 19: Write req - HMI export (indicators) + response handling
            // ============================================================================

            tof_async_write_ind(signal := (par_write_map <> WORD#0) OR (on_demand_write_map <> WORD#0), duration := T#500ms);
            Hmi.s.AsyncWriteIndicator := tof_async_write_ind.output;

            // ============================================================================
            // Network 20: Write acyclic data
            // ============================================================================

            // //Try asynchronous comunication only when synchronous comunication is stable (no errors for 1s)
            // IF (coms_stable) THEN

            //     //Save wr_req value from previous iteation
            //     prev_wr_req := WriteRecord.request;

            //     // React tovalid writes if needed
            //     IF WriteRecord.DONE THEN
            //         Hmi.write_status[async_write_no] := WriteRecord.STATUS;
            //     END_IF;

            //     // Write request error - reset invalidated date if needed
            //     IF WriteRecord.ERROR THEN
            //         Hmi.write_status[async_write_no] := WriteRecord.STATUS;
            //     END_IF;

            //     // Unmask bit map after successfully / unsuccesfully finished write and trigger apropriate re-read
            //     IF (WriteRecord.DONE OR WriteRecord.ERROR) THEN
            //         IF (async_write_no > 0) AND (async_write_no <= 16) THEN
            //             mask := THIS.DECO_WORD(TO_UINT(async_write_no - 1));
            //             par_write_map := par_write_map AND (NOT mask); // unmask the processed write request
            //             par_read_map := par_read_map OR mask; // and request a read to verify/refresh the data
            //         END_IF;
            //         IF (async_write_no > 16) AND (async_write_no <= 32) THEN
            //             mask := THIS.DECO_WORD(TO_UINT(async_write_no - 17));
            //             on_demand_write_map := on_demand_write_map AND (NOT mask); // unmask the processed write request
            //         END_IF;
            //     END_IF;

            //     wr_any_response := (WriteRecord.BUSY OR WriteRecord.DONE OR WriteRecord.ERROR);

            //     //If we get a singnal that request was processed we can set it to false to prepare for generating a new rising edge
            //     IF wr_req AND wr_any_response THEN
            //         wr_req := false;
            //     END_IF;

            //     //If the previous request was processed and we are ready for a new one (new rising edge on rd_req) lets create one
            //     IF Config_async_write_permited AND (NOT prev_wr_req) AND (NOT wr_any_response) AND (NOT coms_just_restored) THEN
            //         IF (par_write_map <> WORD#0) THEN
            //             async_write_no := THIS.ENCO(par_write_map) + 1;
            //             //Fill the write buffer with latest data just before the request
            //             CASE async_write_no OF
            //                 1: //Write buffer 1
            //                     WriteBuffers.buf1.ProcCtrl := Parameters.ProcCtrl;
            //                     WriteBuffers.buf1.ProcLimits := Parameters.ProcLimits;
            //                     WriteBuffers.buf1.FreqCtrl := Parameters.FreqCtrl;
            //                     WriteBuffers.buf1.TriggerByPower := Parameters.TriggerByPower;
            //                     WriteBuffers.buf1.FreqCtrlMode := Parameters.FreqCtrlMode;
            //                     wr_req := true;
            //                 2: //Write buffer 2
            //                     WriteBuffers.buf2.PowerReg := Parameters.PowerReg;
            //                     WriteBuffers.buf2.PressPretrigger := Parameters.PressPretrigger;
            //                     WriteBuffers.buf2.PressTrigger := Parameters.PressTrigger;
            //                     WriteBuffers.buf2.PressTriggerDelay := Parameters.PressTriggerDelay;
            //                     WriteBuffers.buf2.PressWeld := Parameters.PressWeld;
            //                     WriteBuffers.buf2.PressWeldScrub := Parameters.PressWeldScrub;
            //                     WriteBuffers.buf2.PressPostWeld := Parameters.PressPostWeld;
            //                     wr_req := true;
            //                 3: //Write buffer 3
            //                     WriteBuffers.buf3.TriggerTime := Parameters.PressLimits.TriggerTime;
            //                     WriteBuffers.buf3.TriggerPosition := Parameters.PressLimits.TriggerPosition;
            //                     WriteBuffers.buf3.TriggerDelayTime := Parameters.PressLimits.TriggerDelayTime;
            //                     WriteBuffers.buf3.TriggerDelayDistance := Parameters.PressLimits.TriggerDelayDistance;
            //                     WriteBuffers.buf3.Weld1Distance := Parameters.PressLimits.Weld1Distance;
            //                     WriteBuffers.buf3.Weld1Position := Parameters.PressLimits.Weld1Position;
            //                     WriteBuffers.buf3.Weld2Time := Parameters.PressLimits.Weld2Time;
            //                     WriteBuffers.buf3.Weld2Energy := Parameters.PressLimits.Weld2Energy;
            //                     WriteBuffers.buf3.Weld2Power := Parameters.PressLimits.Weld2Power;
            //                     wr_req := true;
            //                 4: //Write buffer 4
            //                     WriteBuffers.buf4.Weld2Distance := Parameters.PressLimits.Weld2Distance;
            //                     WriteBuffers.buf4.Weld2Position := Parameters.PressLimits.Weld2Position;
            //                     WriteBuffers.buf4.TotalWeldTime := Parameters.PressLimits.TotalWeldTime;
            //                     WriteBuffers.buf4.TotalWeldEnergy := Parameters.PressLimits.TotalWeldEnergy;
            //                     WriteBuffers.buf4.TotalWeldDistance := Parameters.PressLimits.TotalWeldDistance;
            //                     WriteBuffers.buf4.DynamicHoldTime := Parameters.PressLimits.DynamicHoldTime;
            //                     WriteBuffers.buf4.DynamicHoldDistance := Parameters.PressLimits.DynamicHoldDistance;
            //                     WriteBuffers.buf4.TotalCycleTime := Parameters.PressLimits.TotalCycleTime;
            //                     WriteBuffers.buf4.FinalHoldPosition := Parameters.PressLimits.FinalHoldPosition;
            //                     WriteBuffers.buf4.ErrorStatus := Parameters.PressLimits.ErrorStatus;
            //                     wr_req := true;

            //                 5: //Write buffer 5
            //                     WriteBuffers.buf5.AnalogSensor := Parameters.AnalogSensor;
            //                     WriteBuffers.buf5.AfterburstEnable := Parameters.AfterburstEnable;
            //                     WriteBuffers.buf5.LimitWeld1TimeEnable := Parameters.LimitWeld1TimeEnable;
            //                     WriteBuffers.buf5.LimitWeld1EnergyEnable := Parameters.LimitWeld1EnergyEnable;
            //                     WriteBuffers.buf5.LimitWeld1PowerEnable := Parameters.LimitWeld1PowerEnable;
            //                     wr_req := true;
            //                 ELSE
            //                     //Unknown parameter write request - just unmask it
            //                     mask := THIS.DECO_WORD(TO_UINT(async_write_no - 1));
            //                     par_write_map := par_write_map AND (NOT mask); // unmask unknown write request
            //                     wr_req := false;
            //                     async_write_no := 0;
            //             END_CASE;
            //         ELSIF (on_demand_write_map <> WORD#0) THEN
            //             async_write_no := THIS.ENCO(on_demand_write_map) + 17;
            //             CASE async_write_no OF
            //                 17: //Copyrec request
            //                     wr_req := true;
            //                 ELSE
            //                     //Unknown on demand write request - just unmask it
            //                     mask := THIS.DECO_WORD(TO_UINT(async_write_no - 17));
            //                     on_demand_write_map := on_demand_write_map AND (NOT mask); // unmask unknown write request
            //                     wr_req := false;
            //                     async_write_no := 0;
            //             END_CASE;
            //         ELSE
            //             //If no request present we call the default WR_REC but without request
            //             async_write_no := 0;
            //         END_IF;
            //     END_IF;

            //     //Safety - if write is not pemited wr_req shoud be always false
            //     IF NOT Config_async_write_permited THEN
            //         wr_req := false;
            //     END_IF;

            //     //Perform the write itself
            //     CASE async_write_no OF
            //         1:  //Write parameter packet 1
            //             THIS.buf1_TO_ByteArray(WriteBuffers.buf1,write_buffer_254);
            //             WriteRecord(request := wr_req,
            //                     id := TO_WORD(Config.HWIDs.HwID_iQ_to_PLC_Inputs),
            //                     index := index_async_data1,
            //                     length := UINT#132,
            //                     record := write_buffer_254);
            //         2:  //Write parameter packet 2
            //             THIS.buf2_TO_ByteArray(WriteBuffers.buf2,write_buffer_254);
            //             WriteRecord(request := wr_req,
            //                     id := TO_WORD(Config.HWIDs.HwID_iQ_to_PLC_Inputs),
            //                     index := index_async_data2,
            //                     length := UINT#136,
            //                     record := write_buffer_254);
            //         3:  //Write parameter packet 3
            //             THIS.buf3_TO_ByteArray(WriteBuffers.buf3,write_buffer_254);
            //             WriteRecord(request := wr_req,
            //                     id := TO_WORD(Config.HWIDs.HwID_iQ_to_PLC_Inputs),
            //                     index := index_async_data3,
            //                     length := UINT#180,
            //                     record := write_buffer_254);
            //         4:  //Write parameter packet 4
            //             THIS.buf4_TO_ByteArray(WriteBuffers.buf4,write_buffer_254);
            //             WriteRecord(request := wr_req,
            //                     id := TO_WORD(Config.HWIDs.HwID_iQ_to_PLC_Inputs),
            //                     index := index_async_data4,
            //                     length := UINT#200,
            //                     record := write_buffer_254);
            //         5:  //Write parameter packet 5
            //             THIS.buf5_TO_ByteArray(WriteBuffers.buf5,write_buffer_254);
            //             WriteRecord(request := wr_req,
            //                     id := TO_WORD(Config.HWIDs.HwID_iQ_to_PLC_Inputs),
            //                     index := index_async_data5,
            //                     length := UINT#176,
            //                     record := write_buffer_254);
            //             //Start of on-demand request types
            //         17: // Copyrec request
            //             write_buffer_254[ 0] := TO_BYTE(SHR(TO_WORD(CopySetup.Destination_Setup),   UINT#8));
            //             write_buffer_254[ 1] := TO_BYTE(    TO_WORD(CopySetup.Destination_Setup));
            //             write_buffer_254[ 2] := TO_BYTE(SHR(TO_WORD(CopySetup.Source_Setup),        UINT#8));
            //             write_buffer_254[ 3] := TO_BYTE(    TO_WORD(CopySetup.Source_Setup));
            //             WriteRecord(request := wr_req,
            //                     id := TO_WORD(Config.HWIDs.HwID_iQ_to_PLC_Inputs),
            //                     index := index_asycn_copyrec,
            //                     length := UINT#4,
            //                     record := write_buffer_254);
            //         ELSE
            //             //By default we call 0 byte WR_REC using REQ=false
            //             THIS.buf1_TO_ByteArray(WriteBuffers.buf1,write_buffer_254);
            //             WriteRecord( request := false,
            //                     id := TO_WORD(Config.HWIDs.HwID_iQ_to_PLC_Inputs),
            //                     index := index_async_data1,
            //                     length := UINT#0,
            //                     record := write_buffer_254);
            //     END_CASE;
            // END_IF;
            // //******************************************

        END_METHOD

        METHOD PUBLIC TemplateMethod_10steps_1 : IAxoTaskState
            TemplateMethod_10steps_1 := TemplateTask_10steps_1.Invoke(THIS);
        END_METHOD

        METHOD PUBLIC TemplateMethod_10steps_2 : IAxoTaskState
            TemplateMethod_10steps_2 := TemplateTask_10steps_2.Invoke(THIS);
        END_METHOD

        METHOD PUBLIC TemplateMethod_10steps_3 : IAxoTaskState
            TemplateMethod_10steps_3 := TemplateTask_10steps_3.Invoke(THIS);
        END_METHOD

        METHOD PUBLIC TemplateMethod_10steps_4 : IAxoTaskState
            TemplateMethod_10steps_4 := TemplateTask_10steps_4.Invoke(THIS);
        END_METHOD

        METHOD PUBLIC TemplateMethod_10steps_5 : IAxoTaskState
            TemplateMethod_10steps_5 := TemplateTask_10steps_5.Invoke(THIS);
        END_METHOD

        METHOD PUBLIC TemplateMethod_10steps_6 : IAxoTaskState
            TemplateMethod_10steps_6 := TemplateTask_10steps_6.Invoke(THIS);
        END_METHOD

        METHOD PUBLIC TemplateMethod_20steps_1 : IAxoTaskState
            TemplateMethod_20steps_1 := TemplateTask_20steps_1.Invoke(THIS);
        END_METHOD

        METHOD PUBLIC TemplateMethod_20steps_2 : IAxoTaskState
            TemplateMethod_20steps_2 := TemplateTask_20steps_2.Invoke(THIS);
        END_METHOD

        METHOD PUBLIC TemplateMethod_20steps_3 : IAxoTaskState
            TemplateMethod_20steps_3 := TemplateTask_20steps_3.Invoke(THIS);
        END_METHOD

        METHOD PUBLIC TemplateMethod_20steps_4 : IAxoTaskState
            TemplateMethod_20steps_4 := TemplateTask_20steps_4.Invoke(THIS);
        END_METHOD

        METHOD PUBLIC TemplateMethod_20steps_5 : IAxoTaskState
            TemplateMethod_20steps_5 := TemplateTask_20steps_5.Invoke(THIS);
        END_METHOD

        METHOD PUBLIC TemplateMethod_20steps_6 : IAxoTaskState
            TemplateMethod_20steps_6 := TemplateTask_20steps_6.Invoke(THIS);
        END_METHOD

        METHOD PROTECTED OVERRIDE ManualControl
            THIS._isManuallyControllable := true;
        END_METHOD

        ///<summary>
        /// Restores this component into intial state.
        ///</summary>
        METHOD PUBLIC OVERRIDE Restore
            VAR
                _index : INT;
            END_VAR
            Status.Action.Id := UINT#0;
            Status.Error.Id  := UINT#0;

            _progress       :=   INT#0;
            _retVal    :=   WORD#0;

            _data_out_1[0] := BYTE#0;
            _data_out_2[0] := BYTE#0;
            _data_out_2[1] := BYTE#0;

            FOR _index := 0 TO 3 DO
                _data_in[_index] := BYTE#0;
                _data_out_4[_index] := BYTE#0;
                _data_out_8[_index] := BYTE#0;
                _data_out_255[_index] := BYTE#0;
            END_FOR;

            FOR _index := 4 TO 7 DO
                _data_in[_index] := BYTE#0;
                _data_out_8[_index] := BYTE#0;
                _data_out_255[_index] := BYTE#0;
            END_FOR;

            FOR _index := 8 TO 254 DO
                _data_in[_index] := BYTE#0;
                _data_out_255[_index] := BYTE#0;
            END_FOR;

            _word           :=   WORD#0;
            _dword          :=   DWORD#0;

            TemplateTask_10steps_1.Restore();
            TemplateTask_10steps_2.Restore();
            TemplateTask_10steps_3.Restore();
            TemplateTask_10steps_4.Restore();
            TemplateTask_10steps_5.Restore();
            TemplateTask_10steps_6.Restore();
            TemplateTask_20steps_1.Restore();
            TemplateTask_20steps_2.Restore();
            TemplateTask_20steps_3.Restore();
            TemplateTask_20steps_4.Restore();
            TemplateTask_20steps_5.Restore();
            TemplateTask_20steps_6.Restore();
            HardwareDiagnosticsTask.Restore();

            Status.Action.Id := UINT#50;
            RestoreTask.DoneWhen(TRUE);

        END_METHOD

        METHOD PRIVATE CallTimers
            VAR_INPUT
                signal : BOOL;
            END_VAR

            _infoTimer.OnDelay(THIS, signal AND Config.InfoTime > T#0S ,Config.InfoTime);
            _errorTimer.OnDelay(THIS, signal AND Config.ErrorTime > T#0S , Config.ErrorTime);

        END_METHOD

    END_CLASS
END_NAMESPACE
